FUNCTION rt_ceild : LREAL
VAR_INPUT
	u: LREAL;
END_VAR
VAR
END_VAR


rt_ceild := DINT_TO_LREAL(TRUNC(u));

IF u = rt_ceild THEN 
    rt_ceild := u;
ELSIF u >= 0.0 THEN 
    rt_ceild := rt_ceild + 1.0;
END_IF;

END_FUNCTION

(* stored: Version 1.1.0.1, ProductVersion 3.1.4024.12
   POU rt_ceild: Id {443fbc25-9d16-40e2-b007-bbb1345740e9}, SpecialFunc None *)
